(* IEC 61131-3 sources: cybercode_codesys_lib/src/signal/Discrete, 5 files *)

(* ---- FB_BasicSignal.st ---- *)
FUNCTION_BLOCK FB_BasicSignal
VAR_INPUT
	ixSignal : BOOL;
END_VAR
VAR_OUTPUT
END_VAR
VAR
END_VAR

METHOD GetInvertedSignal : BOOL
VAR_INPUT
END_VAR
	GetInvertedSignal := NOT ixSignal;
END_METHOD

METHOD GetSignal : BOOL
VAR_INPUT
END_VAR
	GetSignal := ixSignal;
END_METHOD

END_FUNCTION_BLOCK

(* ---- FB_SignalWithFeedback.st ---- *)
FUNCTION_BLOCK FB_SignalWithFeedback EXTENDS FB_BasicSignal
VAR_INPUT
    ixFeedback : BOOL;  	// Сигнал обратной связи
END_VAR
VAR_OUTPUT
END_VAR
VAR
	_inputSignalTrigger : FB_SignalWithTrigger; // Фиксация сигнала поступления команды
	_xWaitingFeedback : BOOL;	// Флаг ожидания сигнала обратной связи
    _xFeedbackReceived : BOOL;  // Флаг успешного получения обратной связи
END_VAR

    _inputSignalTrigger(ixSignal:= GetSignal());

    // Задание флага ожидания сигнала обртаной связи при получении сигнала команды
    IF _inputSignalTrigger.GetRtrig() AND NOT _xWaitingFeedback THEN
        _xWaitingFeedback := TRUE;
    END_IF

    // Задание флага получения обратной связи и ресет флага ожидания
    IF _xWaitingFeedback AND ixFeedback THEN
        _xFeedbackReceived := TRUE;
        ResetWaitingFeedback();
    END_IF

METHOD GetReceivedFeedback : BOOL
VAR_INPUT
END_VAR
    GetReceivedFeedback := _xFeedbackReceived;
END_METHOD

(* Получение статуса флага ожидания сигнала обратной связи*)
METHOD GetWaitingFeedback : BOOL
VAR_INPUT
END_VAR
    GetWaitingFeedback := _xWaitingFeedback;
END_METHOD

METHOD ResetReceivedFeedback
VAR_INPUT
END_VAR
    _xFeedbackReceived := FALSE;
END_METHOD

(* Ресет статуса флага ожидания сигнала обратной связи*)
METHOD ResetWaitingFeedback
VAR_INPUT
END_VAR
    _xWaitingFeedback := FALSE;
END_METHOD

(* ---- FB_SignalWithFeedbackTimer.st ---- *)
FUNCTION_BLOCK FB_SignalWithFeedbackTimer EXTENDS FB_SignalWithFeedback
VAR_INPUT
    tFeedbackTimeout : TIME;  // Время ожидания сигнала обратной связи
END_VAR
VAR_OUTPUT
END_VAR
VAR
    _ton_FeedbackTimeout : TON;  // Таймер ожидания обратной связи
    _xFeedbackTimeout : BOOL;    // Флаг превышения времени ожидания
END_VAR

    // Вызов родительской логики
    SUPER^();

    // Запуск таймера при начале ожидания обратной связи
    _ton_FeedbackTimeout(
        IN := GetWaitingFeedback(),
        PT := tFeedbackTimeout
    );

    // Фиксация ошибки при превышении времени ожидания
    IF _ton_FeedbackTimeout.Q AND NOT _xFeedbackTimeout THEN
        _xFeedbackTimeout := TRUE;
        ResetWaitingFeedback();  // Прекращаем ожидание при таймауте
    END_IF

    // Сброс таймера и ошибки при успешном получении обратной связи
    IF GetReceivedFeedback() THEN
        _ton_FeedbackTimeout(IN := FALSE);
        _xFeedbackTimeout := FALSE;
    END_IF

(* Получение статуса ошибки таймаута обратной связи *)
METHOD GetFeedbackTimeout : BOOL
VAR_INPUT
END_VAR
    GetFeedbackTimeout := _xFeedbackTimeout;
END_METHOD

(* Получение текущего времени ожидания *)
METHOD GetElapsedTime : TIME
VAR_INPUT
END_VAR
    GetElapsedTime := _ton_FeedbackTimeout.ET;
END_METHOD

(* Проверка активности таймера *)
METHOD IsTimerRunning : BOOL
VAR_INPUT
END_VAR
    IsTimerRunning := _ton_FeedbackTimeout.IN;
END_METHOD

(* Сброс ошибки таймаута *)
METHOD ResetFeedbackTimeout
VAR_INPUT
END_VAR
    _xFeedbackTimeout := FALSE;
    _ton_FeedbackTimeout(IN := FALSE);
END_METHOD

(* Полный сброс состояния (включая таймер и ошибки) *)
METHOD Reset
VAR_INPUT
END_VAR
    ResetWaitingFeedback();
    ResetReceivedFeedback();
    ResetFeedbackTimeout();
END_METHOD

END_FUNCTION_BLOCK

(* ---- FB_SignalWithRattling.st ---- *)
FUNCTION_BLOCK FB_SignalWithRattling EXTENDS FB_BasicSignal
VAR_INPUT

END_VAR
VAR_OUTPUT
END_VAR
VAR
    _tStabilityTime : TIME := T#100MS;           // Время стабилизации сигнала
    _nMaxTransitions : UINT := 5;                // Максимальное количество переходов для определения дребезга
    _tDetectionWindow : TIME := T#200MS;         // Окно времени для подсчета переходов

    _ton_StabilityFilter : TON;                 // Таймер фильтрации для стабильного сигнала
    _xOutSignal : BOOL;                         // Отфильтрованный выходной сигнал

    // Переменные для обнаружения дребезга
    _rt_SignalChange : R_TRIG;                  // Детектор фронта 0->1
    _ft_SignalChange : F_TRIG;                  // Детектор фронта 1->0
    _nTransitionCounter : UINT;                 // Счетчик переходов
    _ton_DetectionWindow : TON;                 // Таймер окна обнаружения
    _xRattlingDetected : BOOL;                  // Флаг обнаружения дребезга
    _xPreviousSignal : BOOL;                    // Предыдущее состояние сигнала
    _xDetectionActive : BOOL;                   // Флаг активности обнаружения
END_VAR

// =====================================
// ФИЛЬТРАЦИЯ СИГНАЛА
// =====================================
// Пропускаем сигнал только если он стабилен заданное время
_ton_StabilityFilter(IN := GetSignal(), PT := tStabilityTime);
_xOutSignal := _ton_StabilityFilter.Q;

// =====================================
// ОБНАРУЖЕНИЕ ДРЕБЕЗГА
// =====================================
// Обнаружение изменений сигнала
_rt_SignalChange(CLK := GetSignal());
_ft_SignalChange(CLK := GetSignal());

// Если произошло изменение сигнала
IF _rt_SignalChange.Q OR _ft_SignalChange.Q THEN
    // Если окно обнаружения не активно, запускаем его
    IF NOT _xDetectionActive THEN
        _xDetectionActive := TRUE;
        _nTransitionCounter := 1;  // Первый переход
    ELSE
        // Увеличиваем счетчик переходов
        _nTransitionCounter := _nTransitionCounter + 1;
    END_IF
END_IF

// Таймер окна обнаружения
_ton_DetectionWindow(
    IN := _xDetectionActive,
    PT := tDetectionWindow
);

// Проверка на дребезг в конце окна обнаружения
IF _ton_DetectionWindow.Q THEN
    // Если количество переходов превышает порог - фиксируем дребезг
    IF _nTransitionCounter >= nMaxTransitions THEN
        _xRattlingDetected := TRUE;
    END_IF

    // Сброс окна обнаружения
    _xDetectionActive := FALSE;
    _nTransitionCounter := 0;
    _ton_DetectionWindow(IN := FALSE);
END_IF

// Сохраняем текущее состояние для следующего цикла
_xPreviousSignal := GetSignal();

METHOD GetProcessedSignal : BOOL
VAR_INPUT
END_VAR
    GetProcessedSignal := _xOutSignal;
END_METHOD

(* Получение статуса обнаружения дребезга *)
METHOD GetRattlingDetected : BOOL
VAR_INPUT
END_VAR
    GetRattlingDetected := _xRattlingDetected;
END_METHOD

(* Получение текущего количества переходов в окне обнаружения *)
METHOD GetTransitionCount : UINT
VAR_INPUT
END_VAR
    GetTransitionCount := _nTransitionCounter;
END_METHOD

(* Проверка активности окна обнаружения дребезга *)
METHOD IsDetectionActive : BOOL
VAR_INPUT
END_VAR
    IsDetectionActive := _xDetectionActive;
END_METHOD

(* Получение оставшегося времени окна обнаружения *)
METHOD GetDetectionWindowTime : TIME
VAR_INPUT
END_VAR
    GetDetectionWindowTime := _ton_DetectionWindow.ET;
END_METHOD

(* Сброс ошибки дребезга *)
METHOD ResetRattlingError
VAR_INPUT
END_VAR
    _xRattlingDetected := FALSE;
END_METHOD

(* Полный сброс состояния функционального блока *)
METHOD Reset
VAR_INPUT
END_VAR
    // Сброс ошибки дребезга
    _xRattlingDetected := FALSE;

    // Сброс счетчиков и флагов
    _nTransitionCounter := 0;
    _xDetectionActive := FALSE;

    // Сброс таймеров
    _ton_StabilityFilter(IN := FALSE);
    _ton_DetectionWindow(IN := FALSE);

    // Сброс триггеров
    _rt_SignalChange(CLK := FALSE);
    _ft_SignalChange(CLK := FALSE);

    // Сброс выходного сигнала
    _xOutSignal := FALSE;
END_METHOD

END_FUNCTION_BLOCK

(* ---- FB_SignalWithTrigger.st ---- *)
FUNCTION_BLOCK FB_SignalWithTrigger EXTENDS FB_BasicSignal
VAR_INPUT
END_VAR
VAR_OUTPUT
END_VAR
VAR
	_rt_xSignal : R_TRIG;
	_ft_xSignal : F_TRIG;
END_VAR

    _rt_xSignal(CLK:=GetSignal());
    _ft_xSignal(CLK:= GetSignal());

METHOD GetFtrig : BOOL
VAR_INPUT
END_VAR
    GetFtrig := _ft_xSignal.Q;
END_METHOD

METHOD GetRtrig : BOOL
VAR_INPUT
END_VAR
    GetRtrig := _rt_xSignal.Q;
END_METHOD

END_FUNCTION_BLOCK
